// TIA Portal V20 export
DATA_BLOCK "Sensor"   // DB38
{ S7_Optimized_Access := 'TRUE' }
// stored: MemoryReserve 0
   VAR
      "COMPENSATOR HOMING SENSOR" : Bool;
      "NG & MANUAL INPUT HOMING SENSOR" : Bool;
      "NG & MANUAL INPUT MAGAZINE HOMING SENSOR" : Bool;
      "VISION HOMING SENSOR" : Bool;
      "ELECTRODE NG KICKER HOMING SENSOR" : Bool;
      "CUTTER ROBOT HOMING SENSOR" : Bool;
      "CUTTER HOMING SENSOR" : Bool;
      "ELECTRODE PASS KICKER HOMING SENSOR" : Bool;
      "Tab Sensor" : Bool;
      "Tape Sensor" : Bool;
      "COMPENSATOR LIMIT SENSOR(-)" : Bool;
      "COMPENSATOR LIMIT SENSOR(+)" : Bool;
      "NG & MANUAL INPUT LIMIT SENSOR(-)" : Bool;
      "NG & MANUAL INPUT LIMIT SENSOR(+)" : Bool;
      "NG & MANUAL INPUT MAGAZINE LIMIT SENSOR(-)" : Bool;
      "NG & MANUAL INPUT MAGAZINE LIMIT SENSOR(+)" : Bool;
      "CUTTER ROBOT LIMIT SENSOR(-)" : Bool;
      "CUTTER ROBOT LIMIT SENSOR(+)" : Bool;
      Test_Reset : Bool;
      Test_Timer : TON_TIME;
   END_VAR
BEGIN
END_DATA_BLOCK
